(* IEC 61131-3 sources: stformat/handlers/benchdata, 6 files *)

(* ---- types_and_globals.st ---- *)
{attribute 'qualified_only'}
{attribute 'hide'}

TYPE E_LineState :
	(eStateIdle := 0, eStateRunning := 10, eStateHoming := 20, eStateFault := 99);
END_TYPE

TYPE E_Result :
	(eResultOk := 0, eResultFault := 1, eResultTimeout := 2, eResultBusy := 3);
END_TYPE

TYPE ST_LineStatus :
	STRUCT
		iProduced : INT;
		iRejected : INT;
		fAvailability : LREAL;
		sFault : STRING(80);
		tLastChange : TIME;
		arrStationBusy : ARRAY[1..3] OF BOOL;
	END_STRUCT
END_TYPE

TYPE ST_AxisConfig :
	STRUCT
		fVelocity : LREAL;
		fAcceleration : LREAL;
		fDeceleration : LREAL;
		tTimeout : TIME;
	END_STRUCT
END_TYPE

TYPE ST_Diagnostics :
	UNION
		sText : STRING(32);
		iCode : INT;
		arrWords : ARRAY[0..3] OF WORD;
	END_UNION
END_TYPE

TYPE E_IOQuality :
	INT(0..7);
END_TYPE

TYPE stRecipeEntry :
	STRUCT
		sName : STRING(32);
		fSetpoint : LREAL;
		iFlags : WORD;
	END_STRUCT
END_TYPE

VAR_GLOBAL CONSTANT
	cAXIS_COUNT : INT := 4;
	cDEFAULT_SPEED : LREAL := 250.0;
	cPIPE_DIAMETER : LREAL := 40.0;
	cMAX_CYCLE_MS : UDINT := 250;
	cRecipeSlots : INT := 16;
END_VAR

VAR_GLOBAL
	gAxis : ARRAY[1..cAXIS_COUNT] OF FB_Axis;
	gRecipe : ARRAY[1..cRecipeSlots] OF ST_RecipeEntry;
	gCycleCounter : UDINT;
	gFirstCycleDone : BOOL;
END_VAR

(* ---- diagnostics.st ---- *)
(* Commissioning and diagnostics screen logic. Long argument lists and long
   guard conditions are normal in this code, but they are the exception rather
   than the rule. *)

FUNCTION_BLOCK FB_Diagnostics
VAR_INPUT
	iAxis : INT;
	fPosition : LREAL;
	fTarget : LREAL;
	fVelocity : LREAL;
	bHomed : BOOL;
	bBusy : BOOL;
	nError : INT;
END_VAR

VAR_OUTPUT
	sMessage : STRING(80);
	bAlarm : BOOL;
END_VAR

VAR
	fbStop : MC_Stop;
	fbMoveRelative : MC_MoveRelative;
	tofOvertravel : TOF;
END_VAR

// One long guard: every condition has to hold before a restart is allowed.
IF bHomed
	AND NOT bBusy
	AND nError = 0
	AND ABS(fPosition - fTarget) < 0.05
	AND fVelocity < 0.001
	AND iAxis > 0
	AND iAxis <= cAXIS_COUNT
THEN
	fbStop(bExecute := TRUE, bDecel := TRUE);
	bAlarm := FALSE;
END_IF

tofOvertravel(IN := ABS(fPosition - fTarget) > 1.0, PT := T#2S);
IF tofOvertravel.Q THEN
	fbMoveRelative(
		bExecute := TRUE,
		fDistance := (fTarget - fPosition) * 0.5,
		fVelocity := cDEFAULT_SPEED,
		fAcceleration := cDEFAULT_SPEED,
		fDecel := cDEFAULT_SPEED,
		bRelative := TRUE
	);
	sMessage := CONCAT('Axis ', INT_TO_STRING(iAxis), ' corrected by ', REAL_TO_STRING((fTarget - fPosition) * 0.5));
END_IF

// A full argument list is the other way these lines get long.
fbStop(bExecute := FALSE, bDecel := FALSE, bImmediate := TRUE, fDecel := 0.0, tTimeout := T#0S, bForceAbort := FALSE);
CASE nError OF
	101:
		sMessage := 'Jammed';

	102:
		sMessage := 'Not homed';
	ELSE
		IF bBusy THEN
			sMessage := 'Running';
		END_IF
END_CASE
END_FUNCTION_BLOCK

FUNCTION F_AxisReport : STRING
(160)
VAR_INPUT
	iAxis : INT;
	fPosition : LREAL;
	fTarget : LREAL;
	bHomed : BOOL;
	nError : INT;
END_VAR

IF nError <> 0 THEN
	F_AxisReport := CONCAT('Axis ', INT_TO_STRING(iAxis), ' error ', INT_TO_STRING(nError), ' at ', REAL_TO_STRING(fPosition));
	RETURN;
END_IF

F_AxisReport := CONCAT('Axis ', INT_TO_STRING(iAxis), ' pos ', REAL_TO_STRING(fPosition), ' target ', REAL_TO_STRING(fTarget), ' homed ', BOOL_TO_STRING(bHomed));
END_FUNCTION

(* ---- motion_axis.st ---- *)
(* Motion axis wrapper: profile generator, homing and soft limits. *)

FUNCTION_BLOCK FB_Axis
VAR_INPUT
	bEnable : BOOL;
	fVelocity : LREAL;
	fAcceleration : LREAL;
END_VAR

VAR_OUTPUT
	bBusy : BOOL;
	bDone : BOOL;
	fPosition : LREAL;
	nError : INT;
END_VAR

VAR
	mcMove : MC_MoveAbsolute;
	mcHalt : MC_Halt;
	mcHome : MC_Home;
	bHomed : BOOL;
	fSoftMin : LREAL := - 1000.0;
	fSoftMax : LREAL := 1000.0;
END_VAR

// Soft limits are checked before the command is handed to the axis.
IF fVelocity > 0.0 AND fPosition + (fVelocity * 0.5) > fSoftMax THEN
	nError := 101;
	bBusy := FALSE;
	bDone := TRUE;
	RETURN;
END_IF

IF fVelocity < 0.0 AND fPosition + (fVelocity * 0.5) < fSoftMin THEN
	nError := 102;
	bBusy := FALSE;
	bDone := TRUE;
	RETURN;
END_IF

IF bEnable AND NOT bHomed THEN
	mcHome(
		bExecute := TRUE,
		bClearError := TRUE,
		fHomePosition := 0.0,
		fSpeed := 50.0,
		fAccel := 100.0,
		tTimeout := T#30S
	);
	IF mcHome.bDone THEN
		bHomed := TRUE;
		nError := 0;
	END_IF

	IF mcHome.bError THEN
		nError := mcHome.nErrorID;
	END_IF

	bBusy := mcHome.bBusy;
	bDone := mcHome.bDone;
	RETURN;
END_IF

IF bEnable THEN
	mcMove(
		bExecute := TRUE,
		fTargetPosition := fVelocity,
		fVelocity := fVelocity,
		fAccel := fAcceleration,
		fDecel := fAcceleration,
		bAbsolute := TRUE,
		tTimeout := T#5S
	);
	bBusy := mcMove.bBusy;
	bDone := mcMove.bDone;
	fPosition := mcMove.fActualPosition;
	IF mcMove.bError THEN
		nError := mcMove.nErrorID;
	END_IF

	RETURN;
END_IF

mcHalt(bExecute := TRUE, bDecel := TRUE, fDecel := fAcceleration);
bBusy := mcHalt.bBusy;
bDone := mcHalt.bDone;
fPosition := mcHalt.fActualPosition;
END_FUNCTION_BLOCK

FUNCTION F_Clamp : LREAL
VAR_INPUT
	fValue : LREAL;
	fMinimum : LREAL;
	fMaximum : LREAL;
END_VAR

IF fValue < fMinimum THEN
	F_Clamp := fMinimum;
ELSIF fValue > fMaximum THEN
	F_Clamp := fMaximum;
ELSE
	F_Clamp := fValue;
END_IF
END_FUNCTION

FUNCTION F_DegToRad : LREAL
VAR_INPUT
	fDegrees : LREAL;
END_VAR

F_DegToRad := fDegrees * (PI() / 180.0);
END_FUNCTION

(* ---- numeric.st ---- *)
(* Numeric conversions, literals and time handling. *)

FUNCTION F_Scale : LREAL
VAR_INPUT
	rRaw : INT;
	iRawMin : INT := 0;
	iRawMax : INT := 32767;
	fEngMin : LREAL := 0.0;
	fEngMax : LREAL := 100.0;
END_VAR

VAR
	fSpan : LREAL;
END_VAR

IF iRawMax = iRawMin THEN
	F_Scale := fEngMin;
	RETURN;
END_IF

fSpan := INT_TO_LREAL(iRawMax - iRawMin);
F_Scale := fEngMin + ((INT_TO_LREAL(rRaw) - INT_TO_LREAL(iRawMin)) / fSpan) * (fEngMax - fEngMin);
END_FUNCTION

FUNCTION F_TimeToMs : DWORD
VAR_INPUT
	tValue : TIME;
END_VAR

F_TimeToMs := TIME_TO_DWORD(tValue) / DWORD#1000;
END_FUNCTION

FUNCTION F_BitPattern : DWORD
VAR_INPUT
	byRef : REFERENCE TO BYTE;
	iCount : INT := 4;
END_VAR

VAR
	dwResult : DWORD;
	i : INT;
END_VAR

dwResult := 0;
FOR i := 0 TO iCount - 1 DO
	dwResult := dwResult OR DWORD(SHL(UINT#16, INT_TO_UINT(i)));
END_FOR

F_BitPattern := dwResult;
END_FUNCTION

FUNCTION F_FormatMessage : STRING
(80)
VAR_INPUT
	nCode : INT;
	sDetail : STRING(32);
END_VAR

CASE nCode OF
	1:
		F_FormatMessage := CONCAT('Timeout: ', sDetail);

	2:
		F_FormatMessage := CONCAT('Soft limit: ', sDetail);

	3, 4:
		F_FormatMessage := CONCAT('Axis fault: ', sDetail);

	101:
		F_FormatMessage := CONCAT('Jammed: ', sDetail);

	102:
		F_FormatMessage := 'Not homed';
	ELSE
		F_FormatMessage := sDetail;
END_CASE
END_FUNCTION

FUNCTION_BLOCK FB_TimerBank
VAR_INPUT
	tPeriod : TIME := T#100MS;
END_VAR

VAR_OUTPUT
	arrElapsed : ARRAY[0..7] OF TIME;
	iIndex : INT;
END_VAR

VAR
	ton : ARRAY[0..7] OF TON;
END_VAR

iIndex := iIndex + 1;
IF iIndex > 7 THEN
	iIndex := 0;
END_IF

ton[iIndex](IN := TRUE, PT := tPeriod);
IF ton[iIndex].Q THEN
	arrElapsed[iIndex] := ton[iIndex].ET;
END_IF
END_FUNCTION_BLOCK

FUNCTION F_AddressValid : BOOL
VAR_INPUT
	sAddress : STRING(16);
END_VAR

VAR
	adr : AT %IX0.0;
	p : POINTER TO BYTE;
END_VAR

F_AddressValid := sAddress <> '';
adr.0 := FALSE;
p := ADR(adr);
END_FUNCTION

(* ---- transport_line.st ---- *)
(* Sequence controller for the transport line. *)
(* The machine runs three stations in parallel and hands work between them. *)

FUNCTION_BLOCK FB_TransportLine
VAR_INPUT
	bEnable : BOOL;
	bReset : BOOL;
	tCycleTimeout : TIME := T#10S;
	uiProductCode : UINT;
END_VAR

VAR_OUTPUT
	eState : E_LineState;
	bBusy : BOOL;
	iUnitsProduced : INT;
END_VAR

VAR
	tonCycle : TON;
	tonStation1 : TON;
	tonStation2 : TON;
	tofJam : TOF;
	fbPick : FB_Picker;
	fbPlace : FB_Placer;
	fbConveyor : FB_Conveyor;
	arrStationState : ARRAY[1..3] OF BOOL;
	stStatus : ST_LineStatus;
	iNextStation : INT := 1;
	iRetryCount : INT;
	sLastFault : STRING(80);
END_VAR

VAR CONSTANT
	cMAX_RETRIES : INT := 3;
	cSTATION_COUNT : INT := 3;
END_VAR

METHOD PUBLIC Cycle : BOOL
VAR_INPUT
	bManual : BOOL;
END_VAR

VAR_OUTPUT
	eResult : E_Result;
END_VAR

tonCycle(IN := bEnable, PT := tCycleTimeout);
IF tonCycle.Q THEN
	eResult := eResultTimeout;
	Cycle := FALSE;
	RETURN;
END_IF

IF bReset THEN
	iRetryCount := 0;
	iUnitsProduced := 0;
	sLastFault := '';
	FOR iNextStation := 1 TO cSTATION_COUNT DO
		arrStationState[iNextStation] := FALSE;
	END_FOR

	tonStation1(IN := FALSE);
	tonStation2(IN := FALSE);
	eResult := eResultOk;
	Cycle := TRUE;
	RETURN;
END_IF

// Pick a product and put it on the belt.
fbPick(bEnable := bEnable AND NOT fbConveyor.bFull, iCode := uiProductCode);
IF fbPick.bDone THEN
	iRetryCount := 0;
	fbConveyor(bEnable := TRUE);
END_IF

IF fbConveyor.bFull THEN
	fbPlace(bEnable := TRUE, iTarget := iNextStation);
END_IF

IF fbPlace.bDone THEN
	iUnitsProduced := iUnitsProduced + 1;
	arrStationState[iNextStation] := TRUE;
	iNextStation := iNextStation + 1;
	IF iNextStation > cSTATION_COUNT THEN
		iNextStation := 1;
		eState := eStateIdle;
	END_IF
END_IF

tofJam(IN := NOT fbConveyor.bMoving, PT := T#2S);
IF tofJam.Q THEN
	iRetryCount := iRetryCount + 1;
	sLastFault := CONCAT('Jammed at station ', INT_TO_STRING(iNextStation));
	IF iRetryCount >= cMAX_RETRIES THEN
		eResult := eResultFault;
		eState := eStateFault;
		Cycle := FALSE;
		RETURN;
	END_IF

	tofJam(IN := FALSE);
END_IF

stStatus.iProduced := iUnitsProduced;
stStatus.sFault := sLastFault;
bBusy := eState <> eStateIdle;
eResult := eResultOk;
Cycle := TRUE;
END_METHOD
METHOD PUBLIC Reset : BOOL
VAR
	i : INT;
END_VAR

bReset := TRUE;
fbPick.Reset();
fbPlace.Reset();
fbConveyor.Reset();
FOR i := 1 TO cSTATION_COUNT DO
	arrStationState[i] := FALSE;
END_FOR

Reset := TRUE;
END_METHOD
METHOD PUBLIC GetStatus : ST_LineStatus
VAR_INPUT
	byRef : REFERENCE TO ST_LineStatus;
END_VAR

byRef^ := stStatus;
GetStatus := stStatus;
END_METHOD
PROPERTY PUBLIC UnitsProduced : INT
Get UnitsProduced := iUnitsProduced;
End_Get
END_PROPERTY
END_FUNCTION_BLOCK

(* ---- wiring.st ---- *)
(* Wiring and commissioning helpers. *)

PROGRAM MAIN
VAR
	fbLine : FB_TransportLine;
	fbAxis1 : FB_Axis;
	fbAxis2 : FB_Axis;
	tonStartup : TON;
	iStep : INT;
END_VAR

VAR CONSTANT
	cSTARTUP_DELAY : TIME := T#500MS;
END_VAR

IF gFirstCycleDone THEN
	fbLine(bEnable := TRUE, bReset := FALSE);
END_IF

tonStartup(IN := TRUE, PT := cSTARTUP_DELAY);
IF tonStartup.Q THEN
	fbAxis1(bEnable := TRUE, fVelocity := gRecipe[1].fSetpoint, fAcceleration := cDEFAULT_SPEED);
	fbAxis2(bEnable := FALSE, fVelocity := 0.0, fAcceleration := cDEFAULT_SPEED);
END_IF

CASE iStep OF
	0:
		IF fbLine.bBusy THEN
			iStep := 1;
		END_IF

	1:
		gCycleCounter := gCycleCounter + 1;
		IF fbAxis1.bDone AND fbLine.eState = eStateIdle THEN
			iStep := 0;
		END_IF

	2:
		iStep := 0;
	ELSE
		iStep := 0;
END_CASE
END_PROGRAM

FUNCTION_BLOCK FB_Conveyor
VAR_INPUT
	bEnable : BOOL;
END_VAR

VAR_OUTPUT
	bFull : BOOL;
	bMoving : BOOL;
END_VAR

VAR
	fbAxis : FB_Axis;
	iCount : INT;
END_VAR

fbAxis(bEnable := bEnable, fVelocity := 120.0, fAcceleration := 400.0);
bMoving := fbAxis.bBusy;
bFull := iCount > 20;
iCount := iCount + 1;
END_FUNCTION_BLOCK

FUNCTION_BLOCK FB_Picker
VAR_INPUT
	bEnable : BOOL;
	iCode : UINT;
END_VAR

VAR_OUTPUT
	bDone : BOOL;
END_VAR

REPEAT
	bDone := NOT bEnable;
	EXIT;
UNTIL bDone
END_REPEAT

;
END_FUNCTION_BLOCK

FUNCTION_BLOCK FB_Placer
VAR_INPUT
	bEnable : BOOL;
	iTarget : INT;
END_VAR

VAR_OUTPUT
	bDone : BOOL;
END_VAR

VAR
	i : INT;
END_VAR

i := 0;
WHILE i < 3 AND NOT bDone DO
	i := i + 1;
	bDone := i >= 3;
END_WHILE

;
iTarget := iTarget + 0;
END_FUNCTION_BLOCK
